(* PLC project Programme MGS_2-07_refactorJOY.project, CODESYS CODESYS V3.5 SP19 Patch 1 *)
(* stored: creationDateTime 2026-06-29T23:37:40.3299992, modificationDateTime 2026-06-29T22:49:33.424 *)

FUNCTION_BLOCK FB_Ramp
  VAR_INPUT
    Target : REAL;  (* Cible visée *)
    AccelRate : REAL;  (* Taux d'accélération (%/s) *)
    DecelRate : REAL;  (* Taux de décélération (%/s) *)
    CycleTimeS : REAL;  (* Temps de cycle réel en secondes *)
  END_VAR
  VAR_OUTPUT
    Current : REAL;  (* Valeur courante amortie *)
  END_VAR
  VAR
    StepX : REAL;
  END_VAR

            // Détection du comportement (Accélération vs Décélération)
IF (Target > 0.0 AND Target > Current) OR (Target < 0.0 AND Target < Current) THEN
    StepX := AccelRate * CycleTimeS; // S'éloigne du zéro
ELSE
    StepX := DecelRate * CycleTimeS; // Retourne vers le zéro
END_IF;

// Application de la rampe
IF Current < Target THEN
    Current := Current + StepX;
    IF Current > Target THEN Current := Target; END_IF;
ELSIF Current > Target THEN
    Current := Current - StepX;
    IF Current < Target THEN Current := Target; END_IF;
END_IF;
          
END_FUNCTION_BLOCK
